{attribute 'GeneratedUsingTerminal: EL6201-0000-0017'}
{attribute addProperty BoxType "EL6201-0000-0017"}
{attribute addProperty Id "Slave_25A_DI0BOOL1Slave_25A_DI1BOOL1Slave_25A_DI2BOOL1Slave_25A_DI3BOOL1Slave_25B_DI0BOOL1Slave_25B_DI1BOOL1Slave_25B_DI2BOOL1Slave_25B_DI3BOOL1"}
{attribute addProperty CRC "123371009"}
{attribute addProperty Size "8"}
TYPE Slave_25_Inputs_075A7E01 :
STRUCT
	{attribute addProperty Name "Slave_25A_DI0"}
	Slave_25A_DI0 : BOOL;
	{attribute addProperty Name "Slave_25A_DI1"}
	Slave_25A_DI1 : BOOL;
	{attribute addProperty Name "Slave_25A_DI2"}
	Slave_25A_DI2 : BOOL;
	{attribute addProperty Name "Slave_25A_DI3"}
	Slave_25A_DI3 : BOOL;
	{attribute addProperty Name "Slave_25B_DI0"}
	Slave_25B_DI0 : BOOL;
	{attribute addProperty Name "Slave_25B_DI1"}
	Slave_25B_DI1 : BOOL;
	{attribute addProperty Name "Slave_25B_DI2"}
	Slave_25B_DI2 : BOOL;
	{attribute addProperty Name "Slave_25B_DI3"}
	Slave_25B_DI3 : BOOL;
END_STRUCT
END_TYPE

(* stored: Version 1.2.0.0, ProductVersion 3.1.4024.9
   DUT Slave_25_Inputs_075A7E01: Id {4a9dd9fb-3aa4-49f5-bf5c-a0510dcd87c5} *)
